Yaskawa INFORM job: 01-SAFETY.JBI

/JOB
//NAME 01-SAFETY
///FOLDERNAME SAFETY
//POS
///NPOS 1,1,0,0,0,0
///TOOL 0
///POSTYPE ROBOT
///RECTAN
///RCONF 0,0,0,0,0,0,0,0,0,0,0,0,0,0,0,0,0,0,0,0,0,0,0,0
C00000=1043.969,19.980,-681.842,-3.2680,-33.1635,3.5979
BC00000=539.772,0.033,840.896
//INST
///DATE 2023/07/13 09:06
///ATTR SC,RW,RJ
////FRAME ROBOT
///GROUP1 RB1,BS1
NOP
*START
MOVJ C00000 BC00000 VJ=20.00
JUMP *START
END
